TYPE "A0302_Manager_Ctrl"
VERSION : 0.1
// Block: A0302_Manager_Ctrl
   STRUCT
      EnableStopDoorOpeningReq : Bool;
      EnableStopInPhase : Bool;
      EnableStopProgrammed : Bool;
      Control_ON : Bool;
      REST_Req : Bool;
      WORK_Req : Bool;
      Rest : Bool;
      Work : Bool;
   END_STRUCT;

END_TYPE
